Staubli VAL3: .dtx

mdesc mNomSpeed
sio sioSocket = {link=Socket\toto}
string sTaskPos
string sTaskCmd
string sTaskRobot
jointRx jHere
string sData
num nFrameIndex
num nEol
bool bOvrPosition
num nOvrPos
num nPrevOvrPos
num nSof
num nEof
num nDivider
num nNbChar
num nData
string sDataIn
bool bResult
pointRx pCmdQueue[5]
  [0] = {fatherId=world[0]}
  [1] = {fatherId=world[0]}
  [2] = {fatherId=world[0]}
  [3] = {fatherId=world[0]}
  [4] = {fatherId=world[0]}
num nTypeQueue[5]
num nIndexQueue[5]
num nVelQueue[5]
num nQueueWrite
num nQueueRead
num nQueueCount
num nQueueSize
num nCmdIndex
num nCmdType
num nCmdVel
num nLastIndex
bool bFinish
jointRx jStart
string sAck
num nAckIndex
